TYPE "UDT_ZC_DISP_PPAL_SA"
VERSION : 0.1
   STRUCT
      Orden : Bool;   // Orden activacion
      SegActivacion : Bool;   // Estado seguridad ok
      Consigna : Real;   // Consigna
      ValorActual : Real;   // Valor actual
   END_STRUCT;

END_TYPE

